{attribute addProperty BoxType "EL5032-0000-0021"}
{attribute addProperty Id "StatusAT %I*Status_F504887F1621PositionAT %I*ULINT64817"}
{attribute addProperty CRC "4290005707"}
{attribute addProperty SizeInBites "80"}
{attribute addProperty SizeInBytes "10"}
TYPE FB_Inputs_Channel_FFB44ACB :
STRUCT
	{attribute addProperty Name "Status"}
	Status AT %I* : Status_F504887F;
	{attribute addProperty Name "Position"}
	Position AT %I* : ULINT;
END_STRUCT
END_TYPE

(* stored: Version 1.2.0.0, ProductVersion 3.1.4024.9
   DUT FB_Inputs_Channel_FFB44ACB: Id {633387df-97c6-473d-839f-dec48ffe71a0} *)
